FUNCTION_BLOCK NmGetCfInfo (* Get Connected CFs (intern/extern) *)
  (* Standard: 61499-2 *)
  (* Version 1.0, 2025-09-04, Franz Höpfinger, initial API and implementation and/or initial documentation *)
  PACKAGE isobus::pgn;
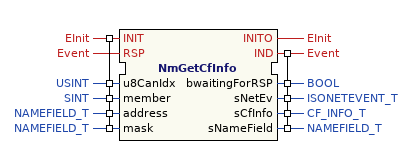
  EVENT_INPUT
    INIT : EInit WITH u8CanIdx, member, address, mask; (* Service Initialization *)
    RSP; (* Response to IND *)
  END_EVENT
  EVENT_OUTPUT
    INITO : EInit; (* Initialization Confirm *)
    IND WITH bwaitingForRSP, sNetEv, sCfInfo, sNameField; (* Indication from Resource *)
  END_EVENT
  VAR_INPUT
    u8CanIdx : USINT := ISO_CAN_NODE::INVALID; (* ISO_CAN_NODE *)
    member : SINT := ISOUSERHOME_e::notdef;
    address : isobus::pgn::NAMEFIELD_T := (bSelfConf := TRUE, bIndGroup := 16#FF, bDevClassInst := 16#FF, bDevClass := 16#FF, bReserved := TRUE, bFunction := 16#FF, bFunctionInst := 16#FF, bEcuInstance := 16#FF, wManufCode := 16#FFFF, dwIdentNumb := 16#FFFFFFFF); (* The Address of the Other Participant *)
    mask : isobus::pgn::NAMEFIELD_T; (* The Mask - only 1 Bits are counted. *)
  END_VAR
  VAR_OUTPUT
    bwaitingForRSP : BOOL; (* the FB is waiting for a RSP now. *)
    sNetEv : isobus::pgn::ISONETEVENT_T; (* network layer event *)
    sCfInfo : isobus::pgn::CF_INFO_T; (* ISO CF/user information data structure *)
    sNameField : isobus::pgn::NAMEFIELD_T; (* ISOBUS Name *)
  END_VAR
END_FUNCTION_BLOCK
